(*			
	RAFALOS
	Rafał Osajda		19.09.2025		TC 4024.66
	Sterowanie językiem systemu
*)
FUNCTION_BLOCK FB_BaseLocation IMPLEMENTS ITF_BaseLocation
VAR
	eLocation		: E_BaseLocation;
	arrLocation		: ARRAY [1..GVL_BaseConstans.LICZBA_DODANYCH_JEZYKOW] OF ST_BaseLocationDesctription := 
						[(wsDescription := "Polski", sCode := 'pl'),
						(wsDescription := "English", sCode := 'en'),
						(wsDescription := "German", sCode := 'de')];;
END_VAR

(*			
	RAFALOS
	Rafał Osajda		24.09.2025		TC 4024.66
	Zwraca kod jezyka tzn 
*)
METHOD PUBLIC GetActualCode : STRING
VAR_INPUT
END_VAR
GetActualCode				:= THIS^.arrLocation [THIS^.eLocation].sCode;
END_METHOD

METHOD PUBLIC GetActualDescription : WSTRING
VAR_INPUT
END_VAR
GetActualDescription			:= THIS^.arrLocation [THIS^.eLocation].wsDescription;
END_METHOD

METHOD PUBLIC GetCode : STRING(5)
VAR_INPUT
	iIN				: INT;
END_VAR
GetCode					:= THIS^.arrLocation [iIN].sCode;
END_METHOD

METHOD PUBLIC GetDescription : WSTRING
VAR_INPUT
	iIN				: INT;
END_VAR
GetDescription				:= THIS^.arrLocation [iIN].wsDescription;
END_METHOD

METHOD PUBLIC GetLocation : E_BaseLocation
VAR_INPUT
END_VAR
GetLocation			:= THIS^.eLocation;
END_METHOD

METHOD PUBLIC SetLocation : BOOL
VAR_INPUT
	sLocation				: STRING;
END_VAR
IF (sLocation = TO_STRING (E_BaseLocation.pl)) THEN
	THIS^.eLocation		:= E_BaseLocation.pl;
	SetLocation			:= TRUE;
ELSIF (sLocation = TO_STRING (E_BaseLocation.en)) THEN
	THIS^.eLocation		:= E_BaseLocation.en;
	SetLocation			:= TRUE;
ELSIF (sLocation = TO_STRING (E_BaseLocation.de)) THEN
	THIS^.eLocation		:= E_BaseLocation.de;
	SetLocation			:= TRUE;
END_IF
END_METHOD

END_FUNCTION_BLOCK

(* stored: Version 1.1.0.1
   POU FB_BaseLocation: Id {3dfcdf37-ccb5-05f1-3cc5-0b09ca33bbd8}, SpecialFunc None
   Method GetActualCode: Id {0792d8a4-a27f-0269-346b-d1f0c252f8f1}
   Method GetActualDescription: Id {055a3d2d-79cd-0f09-0faf-bff15d1193e1}
   Method GetCode: Id {8339f251-4cea-0989-179c-b5279209f3e1}
   Method GetDescription: Id {d5196393-4ada-05db-317f-ff428e81fb58}
   Method GetLocation: Id {fb34d029-b8a1-0ef0-3f71-42e9c3022c0c}
   Method SetLocation: Id {ff1593dc-b625-0ed5-2e8d-1ef6110727ae} *)
